PROGRAM Test
VAR
	unionTest : U_WORD; //unionTest안에 있는 nWord를 값을 넣으면 st16Bit에 nWord값에 맞는 비트로 변함
END_VAR

END_PROGRAM

(* stored: Version 1.1.0.1, ProductVersion 3.1.4026.6
   POU Test: Id {3052891a-721e-4720-be3b-fd81f98127d2}, SpecialFunc None *)
